FUNCTION FC_InitializingSettingLines
VAR_IN_OUT
	HMIInterface	:	MachineSectionHMIInterface;
END_VAR
VAR
	internHMIInterface	:	MachineSectionHMIInterface;
	emptyHMIMovementInterface	:	HMIMovementInterface;
	emptyHMIMovementForkInterface	:	HMIMovementForkInterface;
	emptyHMIRuncontrolInterface	:	HMIRuncontrolInterface;
	emptyHMIRFIDInterface	:	HMIRFIDInterface;
	emptyHMIWorkpieceInterface	:	HMIWorkpieceInterface;
END_VAR

(*===================== Load Interface =====================*)
internHMIInterface := HMIInterface;

(*===================== Initializing Interface =====================*)
internHMIInterface.Movements := emptyHMIMovementInterface;
internHMIInterface.Forks := emptyHMIMovementForkInterface;
internHMIInterface.Runcontrols := emptyHMIRuncontrolInterface;
internHMIInterface.RFID := emptyHMIRFIDInterface;
internHMIInterface.Workpiece := emptyHMIWorkpieceInterface;
(*===================== Write Interface =====================*)
HMIInterface := internHMIInterface;

END_FUNCTION

(* stored: Version 1.1.0.1
   POU FC_InitializingSettingLines: Id {67d42198-5b46-40c6-ab95-402caa5690f2}, SpecialFunc None *)
